// TIA Portal V18 export
TYPE "UDT_AHUsDO"
// stored: IsFailsafeCompliant false
   STRUCT
      xHeaterPumpCmd : Array[1..3] of Bool;
      xSAFAnalogEnable : Array[1..3] of Bool;
      xSAFSp1Cmd : Array[1..3] of Bool;
      xSAFSp2Cmd : Array[1..3] of Bool;
      xCoolerSt1Cmd : Array[1..3] of Bool;
      xCoolerSt2Cmd : Array[1..3] of Bool;
      xCoolerSt3Cmd : Array[1..3] of Bool;
      xCoolerSt4Cmd : Array[1..3] of Bool;
   END_STRUCT;
END_TYPE
